	//OUTPUTS
	bBusy										=> bBusy,
	bComplete									=> bComplete,
	bEnableo									=> bEnableo,
	aPass										=> GVL_HMI_GLOBAL.aGeneralPassHeightTest ,
	aFail										=> GVL_HMI_GLOBAL.aGeneralFailHeightTest ,
	aMinLimitCalibrationBlock					=> stHeightMeasurement2.aMinLimitCalibrationBlock,
	aMaxLimitCalibrationBlock					=> stHeightMeasurement2.aMaxLimitCalibrationBlock,
	aDistanceBetweenProbes						=> stHeightMeasurement2.aDistanceBetweenProbes,
	abSensorStuck								=> stHeightMeasurement2.abSensorStuck,
	nFixedPoint									=> stHeightMeasurement2.nFixedPoint,
	aScaledSensorCurrentValue					=> stHeightMeasurement2.aScaledSensorCurrentValue,
	nHeightMeasureStateValue					=> GVL_HMI_GLOBAL.nHeightMeasureStateValue);

			

IF NOT stStationStruct.bNoCycleStopRequest THEN
	GVL_MASTER.bHeightTestacknowledge := TRUE;
END_IF




//to save data 
GVL_MASTER.stNest.nDistance							:= stHeightMeasurement2.aDistanceBetweenProbes;
GVL_MASTER.stNest.nTarget							:= stHeightMeasurement2.anDistanceSetPoint;
END_ACTION

ACTION ACT_ProbesPosition:
IF ((stHeightMeasurement2.aScaledSensorCurrentValue[1]> GVL_PERSIST.stHeightLimits.nLow)  AND 
	(stHeightMeasurement2.aScaledSensorCurrentValue[1]< GVL_PERSIST.stHeightLimits.nHigh)) AND	
   ((stHeightMeasurement2.aScaledSensorCurrentValue[2]> GVL_PERSIST.stHeightLimits.nLow)  AND 
	(stHeightMeasurement2.aScaledSensorCurrentValue[2]< GVL_PERSIST.stHeightLimits.nHigh)) AND
   ((stHeightMeasurement2.aScaledSensorCurrentValue[3]> GVL_PERSIST.stHeightLimits.nLow)  AND 
	(stHeightMeasurement2.aScaledSensorCurrentValue[3]< GVL_PERSIST.stHeightLimits.nHigh)) AND
   ((stHeightMeasurement2.aScaledSensorCurrentValue[4]> GVL_PERSIST.stHeightLimits.nLow)  AND 
	(stHeightMeasurement2.aScaledSensorCurrentValue[4]< GVL_PERSIST.stHeightLimits.nHigh)) THEN

		GVL_HMI_GLOBAL.bProbesPositionOk				:= TRUE;
ELSE 	GVL_HMI_GLOBAL.bProbesPositionOk				:= FALSE;		
	
END_IF
END_ACTION

ACTION ACT_Statistics:

//GENERAL
IF rtrigCaseTriger[3].Q THEN
GVL_PERSIST.stPartsInspection.nHeightPartsGood:= GVL_PERSIST.stPartsInspection.nHeightPartsGood +1;
GVL_PERSIST.stPartsInspection.nHeightTotalPartsGood := GVL_PERSIST.stPartsInspection.nHeightTotalPartsGood+1;
ELSIF GVL_HMI_GLOBAL.bResetHeightGoodParts THEN
GVL_PERSIST.stPartsInspection.nHeightPartsGood:=0;	
END_IF


IF rtrigCaseTriger[4].Q THEN
	GVL_PERSIST.stPartsInspection.nHeightPartsFailed:=GVL_PERSIST.stPartsInspection.nHeightPartsFailed + 1;
	GVL_PERSIST.stPartsInspection.nHeightTotalPartsFailed:= GVL_PERSIST.stPartsInspection.nHeightTotalPartsFailed + 1;
ELSIF GVL_HMI_GLOBAL.bResetHeightFailParts THEN
	GVL_PERSIST.stPartsInspection.nHeightPartsFailed:=0;
END_IF


//Distance 1

IF rtrigCaseTriger[6].Q THEN
GVL_PERSIST.stPartsInspection.nHeightDistancePartsGood[1]:= GVL_PERSIST.stPartsInspection.nHeightDistancePartsGood[1] +1;
GVL_PERSIST.stPartsInspection.nHeightDistanceTotalPartsGood[1] := GVL_PERSIST.stPartsInspection.nHeightDistanceTotalPartsGood[1]+1;
ELSIF GVL_HMI_GLOBAL.aResetHeightSensorGoodParts[1] THEN
GVL_PERSIST.stPartsInspection.nHeightDistancePartsGood[1]:=0;	
END_IF


IF rtrigCaseTriger[7].Q THEN
	GVL_PERSIST.stPartsInspection.nHeightDistancePartsFailed[1]:=GVL_PERSIST.stPartsInspection.nHeightDistancePartsFailed[1] + 1;
	GVL_PERSIST.stPartsInspection.nHeightDistanceTotalPartsFailed[1]:= GVL_PERSIST.stPartsInspection.nHeightDistanceTotalPartsFailed[1] + 1;
ELSIF GVL_HMI_GLOBAL.aResetHeightSensorBadParts[1] THEN
	GVL_PERSIST.stPartsInspection.nHeightDistancePartsFailed[1]:=0;
END_IF

//Distance 2

IF rtrigCaseTriger[8].Q THEN
GVL_PERSIST.stPartsInspection.nHeightDistancePartsGood[2]:= GVL_PERSIST.stPartsInspection.nHeightDistancePartsGood[2] +1;
GVL_PERSIST.stPartsInspection.nHeightDistanceTotalPartsGood[2] := GVL_PERSIST.stPartsInspection.nHeightDistanceTotalPartsGood[2]+1;
ELSIF GVL_HMI_GLOBAL.aResetHeightSensorGoodParts[2] THEN
GVL_PERSIST.stPartsInspection.nHeightDistancePartsGood[2]:=0;	
END_IF


IF rtrigCaseTriger[9].Q THEN
	GVL_PERSIST.stPartsInspection.nHeightDistancePartsFailed[2]:=GVL_PERSIST.stPartsInspection.nHeightDistancePartsFailed[2] + 1;
	GVL_PERSIST.stPartsInspection.nHeightDistanceTotalPartsFailed[2]:= GVL_PERSIST.stPartsInspection.nHeightDistanceTotalPartsFailed[2] + 1;
ELSIF GVL_HMI_GLOBAL.aResetHeightSensorBadParts[2] THEN
	GVL_PERSIST.stPartsInspection.nHeightDistancePartsFailed[2]:=0;
END_IF

//Distance 3

IF rtrigCaseTriger[10].Q THEN
GVL_PERSIST.stPartsInspection.nHeightDistancePartsGood[3]:= GVL_PERSIST.stPartsInspection.nHeightDistancePartsGood[3] +1;
GVL_PERSIST.stPartsInspection.nHeightDistanceTotalPartsGood[3] := GVL_PERSIST.stPartsInspection.nHeightDistanceTotalPartsGood[3]+1;
ELSIF GVL_HMI_GLOBAL.aResetHeightSensorGoodParts[3] THEN
GVL_PERSIST.stPartsInspection.nHeightDistancePartsGood[3]:=0;	
END_IF


IF rtrigCaseTriger[11].Q THEN
	GVL_PERSIST.stPartsInspection.nHeightDistancePartsFailed[3]:=GVL_PERSIST.stPartsInspection.nHeightDistancePartsFailed[3] + 1;
	GVL_PERSIST.stPartsInspection.nHeightDistanceTotalPartsFailed[3]:= GVL_PERSIST.stPartsInspection.nHeightDistanceTotalPartsFailed[3] + 1;
ELSIF GVL_HMI_GLOBAL.aResetHeightSensorBadParts[3] THEN
	GVL_PERSIST.stPartsInspection.nHeightDistancePartsFailed[3]:=0;
END_IF
END_ACTION

ACTION ACT_TimTrig:
tonCaseDelay[1](IN:= (stStationStruct.nState=300),PT:=T#50MS);
tonCaseDelay[2](IN:= (stStationStruct.nState=1010),PT:=T#100MS);
tonCaseDelay[3](IN:= (stStationStruct.nState=1240),PT:=T#100MS);
tonCaseDelay[4](IN:= ,PT:=T#1S);
tonCaseDelay[5](IN:=stStationStruct.nState=1220 ,PT:=T#2S);
tonCaseDelay[6](IN:= ,PT:=T#250MS);
tonCaseDelay[7](IN:= ,PT:=T#50MS);
tonCaseDelay[8](IN:= ,PT:=T#250MS);
tonCaseDelay[9](IN:= ,PT:=T#250MS);
tonCaseDelay[10](IN:= ,PT:=T#250MS);

rtrigCaseTriger[1](clk:= );
rtrigCaseTriger[2](clk:= );
rtrigCaseTriger[3](clk:= (stStationStruct.nState=1240) AND GVL_MASTER.stNest.bHeightPass );//
rtrigCaseTriger[4](clk:= (stStationStruct.nState=1240) AND NOT GVL_MASTER.stNest.bHeightPass );//
rtrigCaseTriger[5](clk:= stStationStruct.bStationAbort);
rtrigCaseTriger[6](clk:= (stStationStruct.nState=1240) AND GVL_HMI_GLOBAL.aGeneralPassHeightTest[1]);
rtrigCaseTriger[7](clk:= (stStationStruct.nState=1240) AND GVL_HMI_GLOBAL.aGeneralFailHeightTest[1]);
rtrigCaseTriger[8](clk:= (stStationStruct.nState=1240) AND GVL_HMI_GLOBAL.aGeneralPassHeightTest[2]);
rtrigCaseTriger[9](clk:= (stStationStruct.nState=1240) AND GVL_HMI_GLOBAL.aGeneralFailHeightTest[2]);
rtrigCaseTriger[10](clk:= (stStationStruct.nState=1240) AND GVL_HMI_GLOBAL.aGeneralPassHeightTest[3]);
rtrigCaseTriger[11](clk:= (stStationStruct.nState=1240) AND GVL_HMI_GLOBAL.aGeneralFailHeightTest[3]);
END_ACTION

END_PROGRAM

// ---- POUs/G_Utility/FB_HeightMeasurement2.TcPOU
FUNCTION_BLOCK FB_HeightMeasurement2
VAR_INPUT
	
	aSensorCurrentValue							: ARRAY[1..4] OF REAL;		
	bEnable										: BOOL;
	bMeasurementRequest							: BOOL;
	bManualMode									: BOOL;
	bSetFixedPoints								: BOOL;
	aTolerance									: ARRAY[1..3] OF REAL;
	
	bAcknowledge								: BOOL;
	
	//Calibration block
	
	nDistanceBetweenPoints						: ARRAY[1..3] OF REAL;
	anDistanceSetPoint							: ARRAY[1..3] OF REAL;
	
	
	
	
					
END_VAR
VAR_OUTPUT
	
	bBusy										: BOOL;
	bComplete									: BOOL;
	bEnableo									: BOOL;
	aPass										: ARRAY[1..5] OF BOOL; //5 Final Result
	aFail										: ARRAY[1..5] OF BOOL; //5 Final Result
	aMinLimitCalibrationBlock					: ARRAY[1..3] OF REAL;
	aMaxLimitCalibrationBlock					: ARRAY[1..3] OF REAL;
	
	aDistanceBetweenProbes						: ARRAY[1..3] OF REAL; //1 Probe 1 to probe zero
	abSensorStuck								: ARRAY[1..4] OF BOOL;
	nFixedPoint									: ARRAY[1..4] OF REAL;
	aScaledSensorCurrentValue					: ARRAY[1..4] OF REAL;
	
	nHeightMeasureStateValue					: ARRAY[1..4] OF DINT;

	

END_VAR
VAR PERSISTENT
	
	nSensorSetPoint								: ARRAY[1..4] OF REAL;
	
END_VAR
VAR
	
	i											: INT;
	j											: INT;
	tonTestingTime								: TON;
	rMeasurementRequest							: R_TRIG;
	nHeightOffset								: REAL;
	
	EHeighttMeasureProcess						: E_HeighttMeasureProcess;
	anValueBeforeMeasurement					: ARRAY[1..4] OF REAL;
	
	
END_VAR

ACT_ScaleMinMax();
ACT_SetPoints();

IF NOT bEnable THEN
	EHeighttMeasureProcess						:= E_HeighttMeasureProcess.WAITING_ENABLE;
ELSIF bManualMode AND bEnable THEN
	EHeighttMeasureProcess						:= E_HeighttMeasureProcess.Manual_Mode;
END_IF
bEnableo										:= bEnable;
tonTestingTime( IN := (EHeighttMeasureProcess = E_HeighttMeasureProcess.WAITING_FOR_MEASURE), PT := T#3S);
rMeasurementRequest( CLK := bMeasurementRequest);

CASE EHeighttMeasureProcess OF

E_HeighttMeasureProcess.WAITING_ENABLE:

	IF bEnable THEN
		EHeighttMeasureProcess					:= E_HeighttMeasureProcess.WAITING_MEASURING_REQUEST;
	END_IF

E_HeighttMeasureProcess.WAITING_MEASURING_REQUEST:	

	bComplete									:= FALSE;
	IF rMeasurementRequest.Q THEN
		EHeighttMeasureProcess					:= E_HeighttMeasureProcess.RESET;
	END_IF
	
	anValueBeforeMeasurement					:= aSensorCurrentValue;

E_HeighttMeasureProcess.RESET:
	
	
	abSensorStuck[1]							:= FALSE;
	
	FOR i := 1 TO 5 DO
		aPass[i]								:= FALSE;	
		aFail[i]								:= FALSE;
	END_FOR
	FOR j := 1 TO 3 DO
		nHeightMeasureStateValue[j]				:= 0;
	END_FOR
		EHeighttMeasureProcess					:= E_HeighttMeasureProcess.WAITING_FOR_MEASURE;
	
E_HeighttMeasureProcess.SENSOR_STUCK_EVALUATION:

	ACT_SensorStuck();
	
E_HeighttMeasureProcess.WAITING_FOR_MEASURE:

	IF tonTestingTime.Q  THEN
		EHeighttMeasureProcess					:= E_HeighttMeasureProcess.CALIBRATIONBLOCK_METHOD;
	END_IF

E_HeighttMeasureProcess.CALIBRATIONBLOCK_METHOD:

		ACT_CalibrationBlockMethod();
		bComplete								:= TRUE;
		IF bAcknowledge THEN
			EHeighttMeasureProcess					:= E_HeighttMeasureProcess.WAITING_MEASURING_REQUEST;
		END_IF

E_HeighttMeasureProcess.Manual_Mode:
		
		ACT_ManualMode();		

END_CASE


bBusy				:= 	(EHeighttMeasureProcess	<> E_HeighttMeasureProcess.WAITING_ENABLE AND
						EHeighttMeasureProcess  <> E_HeighttMeasureProcess.WAITING_MEASURING_REQUEST) AND
						NOT bComplete;

ACTION ACT_CalibrationBlockMethod:
aDistanceBetweenProbes[1] 	:= (nFixedPoint[4] - aScaledSensorCurrentValue[4])+ (aScaledSensorCurrentValue[1] - (nFixedPoint[1])) + nDistanceBetweenPoints[1];
aDistanceBetweenProbes[2] 	:= (nFixedPoint[4] - aScaledSensorCurrentValue[4])+ (aScaledSensorCurrentValue[2] - (nFixedPoint[2])) + nDistanceBetweenPoints[2];
aDistanceBetweenProbes[3] 	:= (nFixedPoint[4] - aScaledSensorCurrentValue[4])+ (aScaledSensorCurrentValue[3] - (nFixedPoint[3])) + nDistanceBetweenPoints[3];

FOR i := 1 TO 3 DO
	IF (aDistanceBetweenProbes[i] <= aMaxLimitCalibrationBlock[i]) AND (aDistanceBetweenProbes[i] >= aMinLimitCalibrationBlock[i]) THEN
		
		aPass[i]			:= TRUE;
		nHeightMeasureStateValue[i] := 1;
	ELSE 
		aFail[i]			:= TRUE;
		nHeightMeasureStateValue[i] := 2;
	END_IF
END_FOR

IF aPass[1] AND aPass[2] AND aPass[3] THEN
	aPass[5]			:= TRUE;
ELSIF aFail[1] OR aFail[2] OR aFail[3] THEN
	aFail[5]			:= TRUE;
END_IF
END_ACTION

ACTION ACT_ManualMode:
aDistanceBetweenProbes[1] 	:= (nFixedPoint[4] - aScaledSensorCurrentValue[4])+ (aScaledSensorCurrentValue[1] - (nFixedPoint[1])) + nDistanceBetweenPoints[1];
aDistanceBetweenProbes[2] 	:= (nFixedPoint[4] - aScaledSensorCurrentValue[4])+ (aScaledSensorCurrentValue[2] - (nFixedPoint[2])) + nDistanceBetweenPoints[2];
aDistanceBetweenProbes[3] 	:= (nFixedPoint[4] - aScaledSensorCurrentValue[4])+ (aScaledSensorCurrentValue[3] - (nFixedPoint[3])) + nDistanceBetweenPoints[3];

IF (aDistanceBetweenProbes[1] <= aMaxLimitCalibrationBlock[1]) AND (aDistanceBetweenProbes[1] >= aMinLimitCalibrationBlock[1]) THEN
	
		nHeightMeasureStateValue[1] := 1;
ELSE 
		nHeightMeasureStateValue[1] := 2;
END_IF

IF (aDistanceBetweenProbes[2] <= aMaxLimitCalibrationBlock[2]) AND (aDistanceBetweenProbes[2] >= aMinLimitCalibrationBlock[2]) THEN
	
		nHeightMeasureStateValue[2] := 1;
ELSE 
		nHeightMeasureStateValue[2] := 2;
END_IF

IF (aDistanceBetweenProbes[3] <= aMaxLimitCalibrationBlock[3]) AND (aDistanceBetweenProbes[3] >= aMinLimitCalibrationBlock[3]) THEN
	
		nHeightMeasureStateValue[3] := 1;
ELSE 
		nHeightMeasureStateValue[3] := 2;
END_IF
END_ACTION

ACTION ACT_ScaleMinMax:
//Current value SCALE
IF aSensorCurrentValue[1] <> 0 THEN
	
	aScaledSensorCurrentValue[1]		:= aSensorCurrentValue[1]/10000;
	
ELSE aScaledSensorCurrentValue[1]		:= 0;

END_IF

IF aSensorCurrentValue[2] <> 0 THEN
	
	aScaledSensorCurrentValue[2]		:= aSensorCurrentValue[2]/10000;
	
ELSE aScaledSensorCurrentValue[2]		:= 0;

END_IF

IF aSensorCurrentValue[3] <> 0 THEN
	
	aScaledSensorCurrentValue[3]		:= aSensorCurrentValue[3]/10000;
	
ELSE aScaledSensorCurrentValue[3]		:= 0;

END_IF

IF aSensorCurrentValue[4] <> 0 THEN
	
	aScaledSensorCurrentValue[4]		:= aSensorCurrentValue[4]/10000;
	
ELSE aScaledSensorCurrentValue[4]		:= 0;

END_IF

aMaxLimitCalibrationBlock[1]			:= anDistanceSetPoint[1] + aTolerance[1];
aMaxLimitCalibrationBlock[2]			:= anDistanceSetPoint[2] + aTolerance[2];
aMaxLimitCalibrationBlock[3]			:= anDistanceSetPoint[3] + aTolerance[3];

aMinLimitCalibrationBlock[1]			:= anDistanceSetPoint[1] - aTolerance[1];
aMinLimitCalibrationBlock[2]			:= anDistanceSetPoint[2] - aTolerance[2];
aMinLimitCalibrationBlock[3]			:= anDistanceSetPoint[3] - aTolerance[3];
END_ACTION

ACTION ACT_SensorStuck:
IF (anValueBeforeMeasurement[1] <= (aSensorCurrentValue[1] + 0.5)) AND (anValueBeforeMeasurement[1] >= (aSensorCurrentValue[1] - 0.5)) THEN
		abSensorStuck[1]							:= TRUE;
	END_IF

IF (anValueBeforeMeasurement[2] <= (aSensorCurrentValue[2] + 0.5)) AND (anValueBeforeMeasurement[2] >= (aSensorCurrentValue[2] - 0.5)) THEN
		abSensorStuck[2]							:= TRUE;
	END_IF

IF (anValueBeforeMeasurement[3] <= (aSensorCurrentValue[3] + 0.5)) AND (anValueBeforeMeasurement[3] >= (aSensorCurrentValue[3] - 0.5)) THEN
		abSensorStuck[3]							:= TRUE;
	END_IF

IF (anValueBeforeMeasurement[4] <= (aSensorCurrentValue[4] + 0.5)) AND (anValueBeforeMeasurement[4] >= (aSensorCurrentValue[4] - 0.5)) THEN
		abSensorStuck[4]							:= TRUE;
	END_IF
END_ACTION

ACTION ACT_SetPoints:
IF bSetFixedPoints THEN
	
	nSensorSetPoint[1]						:= aScaledSensorCurrentValue[1];
	nSensorSetPoint[2]						:= aScaledSensorCurrentValue[2];
	nSensorSetPoint[3]						:= aScaledSensorCurrentValue[3];
	nSensorSetPoint[4]						:= aScaledSensorCurrentValue[4];
ELSE
	
	nFixedPoint[1]							:= nSensorSetPoint[1];
	nFixedPoint[2]							:= nSensorSetPoint[2];
	nFixedPoint[3]							:= nSensorSetPoint[3];
	nFixedPoint[4]							:= nSensorSetPoint[4];



END_IF
END_ACTION

END_FUNCTION_BLOCK
